// TIA Portal project "Ejemplo_3" (V16)

(* hardware
DEVICE "S7300/ET200M station_1"  S7-300 station
   slot 0: "Perfil soporte_0"  Rail  6ES7 390-1***0-0AA0
   slot 2: "PLC_1"  CPU 313C  6ES7 313-5BG04-0AB0  V3.3
      slot 0: "Interfaz MPI_1"  MPI
      slot 2: "DI 24/DO 16_1"  DI24/DO16
      slot 3: "AI 5/AO 2_1"  AI5/AO2
      slot 4: "Contaje_1"  Counter
*)

// ===== PLC "PLC_1"  CPU 313C =====

VAR_GLOBAL   // PLC tag table "Tabla de variables estándar"
   "Mem_Acu" AT %MW1 : Int;
   "Tag_1" AT %M0.0 : Bool;
   "Tag_2" AT %I124.0 : Bool;
END_VAR

DATA_BLOCK "Bloque_1_DB"   // DB1
{ S7_Optimized_Access := 'FALSE' }
VERSION : 0.1
// stored: InstanceOfName Bloque_1
"Bloque_1"
BEGIN
END_DATA_BLOCK

FUNCTION_BLOCK "Bloque_1"   // FB1, LAD
{ S7_Optimized_Access := 'FALSE' }
VERSION : 0.1
   VAR
      Acumulador : Int;
   END_VAR
BEGIN

REGION Network 1
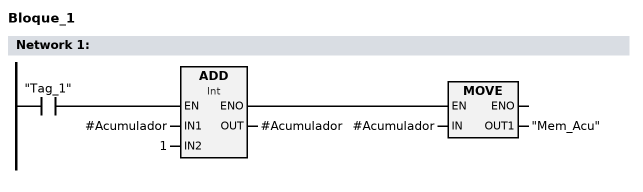
   RUNG wire#powerrail
      Contact( "Tag_1" )
      { S7_Templates := "SrcType := Int"; S7_GenerateENO := "TRUE" } Add(in1 := #Acumulador, in2 := 1, out => #Acumulador)
      { S7_GenerateENO := "TRUE" } Move(in := #Acumulador, out1 => "Mem_Acu")
   END_RUNG
   // the same network as SCL:
   // ENO of a box is taken as its EN; it also drops when the box reports an error
   IF "Tag_1" THEN
       #Acumulador := #Acumulador + 1;
       "Mem_Acu" := #Acumulador;
   END_IF;
END_REGION
END_FUNCTION_BLOCK

FUNCTION "Bloque_2" : Void   // FC1, LAD
{ S7_Optimized_Access := 'FALSE' }
VERSION : 0.1
   VAR_TEMP
      Acumulador : Int;
   END_VAR
BEGIN

REGION Network 1
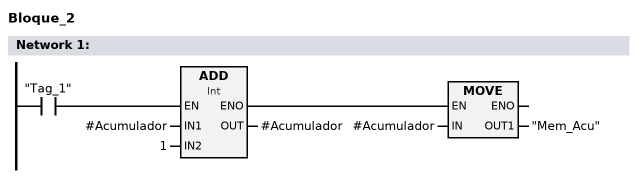
   RUNG wire#powerrail
      Contact( "Tag_1" )
      { S7_Templates := "SrcType := Int"; S7_GenerateENO := "TRUE" } Add(in1 := #Acumulador, in2 := 1, out => #Acumulador)
      { S7_GenerateENO := "TRUE" } Move(in := #Acumulador, out1 => "Mem_Acu")
   END_RUNG
   // the same network as SCL:
   // ENO of a box is taken as its EN; it also drops when the box reports an error
   IF "Tag_1" THEN
       #Acumulador := #Acumulador + 1;
       "Mem_Acu" := #Acumulador;
   END_IF;
END_REGION
END_FUNCTION

ORGANIZATION_BLOCK "Main"   // OB1, LAD
TITLE = "Main Program Sweep (Cycle)"
{ S7_Optimized_Access := 'FALSE' }
VERSION : 0.1
   VAR_TEMP
      OB1_EV_CLASS : Byte;   // Bits 0-3 = 1 (Coming event), Bits 4-7 = 1 (Event class 1)
      OB1_SCAN_1 : Byte;   // 1 (Cold restart scan 1 of OB 1), 3 (Scan 2-n of OB 1)
      OB1_PRIORITY : Byte;   // Priority of OB Execution
      OB1_OB_NUMBR : Byte;   // 1 (Organization block 1, OB1)
      OB1_RESERVED_1 : Byte;   // Reserved for system
      OB1_RESERVED_2 : Byte;   // Reserved for system
      OB1_PREV_CYCLE : Int;   // Cycle time of previous OB1 scan (milliseconds)
      OB1_MIN_CYCLE : Int;   // Minimum cycle time of OB1 (milliseconds)
      OB1_MAX_CYCLE : Int;   // Maximum cycle time of OB1 (milliseconds)
      OB1_DATE_TIME : Date_And_Time;   // Date and time OB1 started
   END_VAR
BEGIN

REGION Network 1
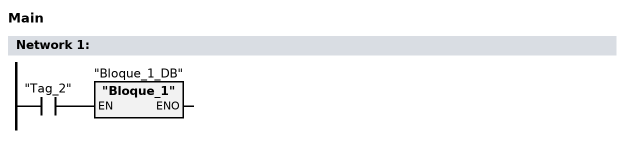
   RUNG wire#powerrail
      Contact( "Tag_2" )
      "Bloque_1_DB"()
   END_RUNG
   // the same network as SCL:
   IF "Tag_2" THEN
       "Bloque_1_DB"();   // "Bloque_1"
   END_IF;
END_REGION
END_ORGANIZATION_BLOCK